TYPE EL9220ChannelInput :
STRUCT
    status AT AT%I* : EL9220StatusInput;
    load AT AT%I* : UINT;
    current AT AT%I* : UINT;
    voltagIn AT AT%I* : UINT;
    voltageOut AT AT%I* : UINT;
END_STRUCT
END_TYPE

(* stored: Version 1.1.0.1, ProductVersion 3.1.4020.12
   DUT EL9220ChannelInput: Id {5dd48cb9-7874-4e81-8f40-14fca077ddd2} *)
